TYPE U_Convert :
UNION
	AsWord: ARRAY[0..1] OF WORD;
	AsReal: REAL;
END_UNION
END_TYPE

(* stored: Version 1.1.0.1
   DUT U_Convert: Id {aaf5a80a-4fff-42cd-a217-146edfe0780d} *)
